Universal Robots PolyScope program: quality_ccc.urp

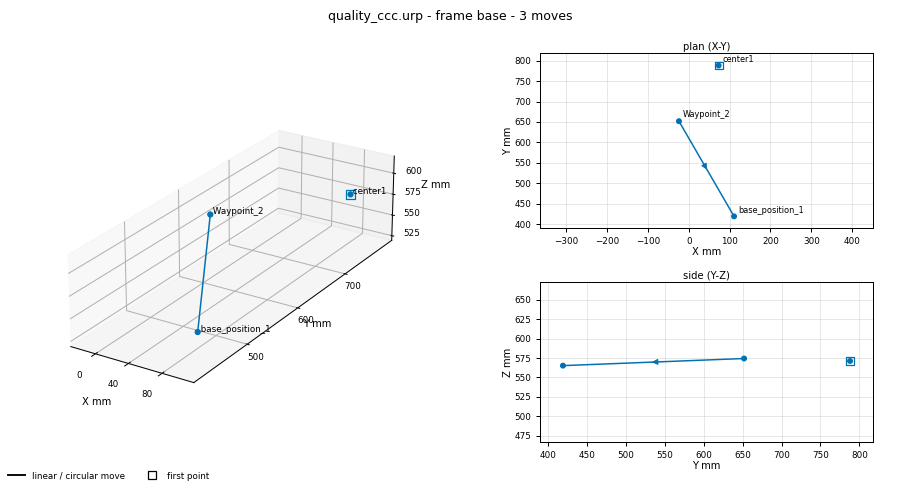
[picture p0: tool path of quality_ccc.urp in frame base, 3 of 9 moves have a stored position in this frame; points joined in program order, loops and branches not executed]
Program quality_ccc (installation=default directory=/programs/Nicolas_Arteaga/quality createdIn=5.8.2.10297 lastSavedIn=5.12.4.1101661 robotSerialNumber=20225502378)
Calibrated DH parameters: a=[0.00022, -0.425328, -0.389701, 0.000059, 0.000065, 0]; d=[0.162608, 0.803456, 9.992211, -10.662202, 0.099702, 0.099559]; alpha=[1.570756, 0.001543, 0.004316, 1.570651, -1.570122, 0]; deltaTheta=[0, 0.002917, 0.116094, -0.119008, 0, -0.000001]
Robot Program (runOnlyOnce=true)
  MoveJ speed 60 deg/s, acceleration 80 deg/s^2 (useActiveTCP=true) feature=Base
    Waypoint center1: TCP in base x=73.068 y=788.065 z=571.167 mm, rx=-1.5688 ry=-0.0203 rz=0.0146 rad; joints [245.634, -75.761, 61.592, 13.883, 64.245, 180.144] deg; TCP offset x=0 y=0 z=191.5 mm, rx=0 ry=0 rz=0 rad
  'Now Cotton Candy Creation'
  SuppressedNode
    radius := 0.149
  radius := 0.135
  height := 0.05
  SuppressedNode
    cold_start_wait := 101.25
  SuppressedNode
    wait_time := GP_int_in[1]
  wait_time := 0
  cook_time := GP_int_in[2]
  SuppressedNode
    circle_time := GP_int_in[2]
  SuppressedNode
    wait_time := 1
  SuppressedNode
    cook_time := 33.75
  circle_time := 3.75
  SuppressedNode
    cold_start_spin := 28
  SuppressedNode
    cold_start_spin := 100
  center := Joint_6_name
  bottom := pose_add(center, p[0, -radius, height, 0, 0, 0])
  right := pose_add(center, p[-radius, 0, -height, 0, 0, 0])
  top_circ := pose_add(center, p[0, radius, height, 0, 0, 0])
  left := pose_add(center, p[radius, 0, -height, 0, 0, 0])
  SuppressedNode
    diff := pose_sub(left,bottom )
  SuppressedNode
    Loop While (checkContinuously=false) expression=circles_no>0
      MoveP speed 250 mm/s, acceleration 1200 mm/s^2 (blendRadius=0.125 useActiveTCP=true) feature=Base
        Waypoint Waypoint (Variable): variable=bottom
        CircleMove (OrientationMode=UNCONSTRAINED)
          Waypoint Waypoint (Variable): variable=left
          Waypoint Waypoint (Variable): variable=top_circ
      MoveP speed 250 mm/s, acceleration 1200 mm/s^2 (blendRadius=0.025 useActiveTCP=true) feature=Base
        Waypoint Waypoint (Variable): variable=top_circ
        CircleMove (OrientationMode=UNCONSTRAINED)
          Waypoint Waypoint (Variable): variable=right
          Waypoint Waypoint (Variable): variable=bottom
      circles_no := circles_no-1
  SuppressedNode
    Timer (action=Stop) variable(name=timer_3)
  SuppressedNode
    Wait Sleep waitTime=101.25
  SuppressedNode
    Wait Condition expression=GP_int_in[0]
  Script: sleep(wait_time)
  Timer (action=Start) variable(name=timer_1)
  Loop While (checkContinuously=false) expression=cook_time>0
    MoveP speed 250 mm/s, acceleration 1200 mm/s^2 (blendRadius=0.125 useActiveTCP=true) feature=Base
      Waypoint Waypoint (Variable): variable=bottom
      CircleMove (OrientationMode=UNCONSTRAINED)
        Waypoint Waypoint (Variable): variable=left
        Waypoint Waypoint (Variable): variable=top_circ
    MoveP speed 250 mm/s, acceleration 1200 mm/s^2 (blendRadius=0.025 useActiveTCP=true) feature=Base
      Waypoint Waypoint (Variable): variable=top_circ
      CircleMove (OrientationMode=UNCONSTRAINED)
        Waypoint Waypoint (Variable): variable=right
        Waypoint Waypoint (Variable): variable=bottom
    cook_time := cook_time-circle_time
  MoveL speed 250 mm/s, acceleration 1200 mm/s^2 (useActiveTCP=true) feature=Base
    Waypoint Waypoint_2: TCP in base x=-24.03 y=651.793 z=574.352 mm, rx=-0.9882 ry=-1.0644 rz=-1.2372 rad; joints [248.909, -99.854, 96.502, -11.42, 64.977, 96.89] deg
    Waypoint base_position_1: TCP in base x=110.843 y=418.879 z=565.205 mm, rx=-1.5601 ry=-0.9892 rz=-1.3624 rad; joints [201.946, -128.865, 99.355, 35.834, 42.385, 90.241] deg
